// TIA Portal V20 export
DATA_BLOCK "EmData"   // DB92
// stored: Access Published, MemoryReserve 100, Namespace Unit1
   VAR
      anodeElectrode : DInt;
      cathodeElectrode : DInt;
      currentTotalElectrode : DInt;
      targetTotalElectrode : DInt := 39;
      oldTotalElectrode : DInt;
      remainValue : DInt;   // Return reminder of divison.
      cpm : DInt := 80;
      homing : Bool;
      PartData : Struct
         EM4 : "LER_typePartDataEm4";
         EM5 : "LER_typePartDataEm5";
         EM6 : "LER_typePartDataEm6";
         EM7 : "LER_typePartDataEm7";
         clearPartData : "LER_typePartData";
         clearTableBuffer : Array[0..59] of "LER_typeUnitData";
      END_STRUCT;
   END_VAR
   VAR RETAIN
      PartData_Move : Array[0..10] of "LER_typePartData";
   END_VAR
   VAR
      calculateResult : Struct
         sepaClampCutterAxisX { S7_SetPoint := 'True'} : "LBC_typeAxis64PosConfiguration";
         sepaClampCutterAxisZ { S7_SetPoint := 'True'} : "LBC_typeAxis64PosConfiguration";
         sepaGripperAxisX { S7_SetPoint := 'True'} : "LBC_typeAxis64PosConfiguration";
         pusherAxisZ { S7_SetPoint := 'True'} : "LBC_typeAxis64PosConfiguration";
      END_STRUCT;
      UnitRecipe : Struct
         size : "LER.Size";
         SepaThickness { S7_SetPoint := 'True'} : LReal := 0.25;
         JellyRollWidth : LReal;
         StackCount : DInt := 39;
         DancerRegulator : LReal;
         AutoSpliceRemainingLength : LReal;
         TotalSepaWebLenth : LReal;
      END_STRUCT;
      TEST : Array[0..99] of Bool;
      RunOutModeControl : Struct   // Run Out Mode Start
         RunOutStart : Bool;
         RunOutComplete : Bool;
      END_STRUCT;
   END_VAR
   VAR RETAIN
      DataBit : Struct
         AnodePnP1 : Bool;
         AnodePnP2 : Bool;
         AnodeTable : Bool;
         CathodePnP1 : Bool;
         CathodePnP2 : Bool;
         CathodeTable : Bool;
      END_STRUCT;
   END_VAR
BEGIN
   // PartData_Move[1] : AnodeMainPnP1
   // PartData_Move[2] : AnodeAlignTable
   // PartData_Move[3] : AnodeMainPnP2
   // PartData_Move[4] : StackTable
   // PartData_Move[5] : CathodeMainPnP2
   // PartData_Move[6] : CathodeAlignTable
   // PartData_Move[7] : CathodeMainPnP1
   // PartData_Move[8] : Winder
   // PartData_Move[9] : SepaGripper
   calculateResult.sepaClampCutterAxisX.setPositions[3]."name" := 'Angle90';
   calculateResult.sepaClampCutterAxisX.setPositions[4]."name" := 'Angle180';
   calculateResult.sepaClampCutterAxisX.setPositions[5]."name" := 'Angle270';
   calculateResult.sepaClampCutterAxisX.setPositions[6]."name" := 'Angle360';
   calculateResult.pusherAxisZ.setPositions[2]."name" := 'VerticalPos';
   calculateResult.pusherAxisZ.setPositions[3]."name" := 'HorizonPos';
   UnitRecipe.size.Anode.thickness := 0.5;
   UnitRecipe.size.Anode.length := 200.0;
   UnitRecipe.size.Cathode.thickness := 0.5;
   UnitRecipe.size.Cathode.length := 200.0;
   // TEST[0] : Anode Align Vision NG
   // TEST[1] : Anode Align Vision OK
   // TEST[2] : Cathode Align Vision NG
   // TEST[3] : Cathode Align Vision OK
   // TEST[4] : Stack Table Gap Vision NG
   TEST[5] := TRUE;   // Stack Table Gap Vision OK
   // TEST[10] : HMI Anode NG Data Generate Button
   // TEST[11] : HMI Cathode NG Data Generate Button
   // TEST[13] : Stack Main Ready Stop Requset
END_DATA_BLOCK
